PROGRAM MAIN
VAR
		
	bAllDone		: BOOL;
	bStopSequence	: BOOL;
	
	nCase 		: INT;
	nMoveState		: ARRAY[1..nNumMaxMovers] OF INT;
	
	aDynamics	: ARRAY[1..nNumMaxMovers] OF DynamicConstraint_PathXY;
	aMoveOnTrackOptions : ARRAY[1..20] OF ST_MoveOnTrackOptions;
	
	fbXtsEnvironment: FB_TcIoXtsEnvironment;
	
	nForCounter: UDINT;
	M,N,T,Tr,i : UDINT;
	dynamics: INT;
	
	// Magnet
	MagnetValue AT%Q*: INT;
	bMagnetOn : BOOL;	
	stPositionInfo: ST_PositionInfo;
		
	pwm: FB_PWM;
	
	IsMoverCommandedInShortcut: BOOL;
	IsMoverInBlockingArea: BOOL;
	nActStopPos: UINT := 1;
	Fp_error : R_Trig;
	Velo : LREAL := 500;
	Velom1 : LREAL := 500;
	Switch : BOOL;
	WithoutSwitch : BOOL;
	SwtichOnly: BOOL;
	
	MoverStop 		AT%I* : BOOL;
	MoverStopDone 	AT%Q* : BOOL;
	Info 			AT%Q* : BOOL;
	Operating		AT%Q* : BOOL;
	Process			AT%Q* : BOOL;
	Fault			AT%Q* : BOOL;
	Emergency		AT%Q* : BOOL;
	
	Voltage1 		AT%I* : UDINT;
	Voltage2 		AT%I* : UDINT;
	
	
	TcRestart : TC_Restart;
	Restart : BOOL;
	busy : BOOL;
	fp_start : R_Trig;
	bStartSequence: BOOL;
	
	FP_Counter : r_trig;
	Switchcounter : DINT;
	SwitchCurrent: INT :=12; 
	test : LREAL;
	Horntimer : tp; 
	R_trigHorn : R_trig;
	
	TestPowerMat : BOOL;
	StopPos : LREAL := 7611;
	StopTime : TIME := T#8S;
	StopTimer :ARRAY[1..nNumMaxMovers] OF ton;
	StartTimer :ARRAY[1..nNumMaxMovers] OF BOOL;
	
	
	MoverPos :ARRAY[1..nNumMaxMovers] OF PositionXYC;
	ArcLength :ARRAY[1..nNumMaxMovers] OF LREAL;
	TrackPos :ARRAY[1..nNumMaxMovers] OF ARRAY[1..nNumMaxTracks] OF PositionXYC;
	fbFlashlight : Flashlight;
END_VAR

fbXtsEnvironment.Init(TRUE);

Emergency := NOT  MoverStop;


R_trigHorn(clk := MoverStop);
Horntimer(in:= ( R_trigHorn.Q ) , PT:= T#5S,Q=> info);
fbFlashlight(Frequence:=5 , Error=> , Blinker=> );

IF  NOT Horntimer.Q AND MoverStop THEN
	Process := TRUE;
ELSIF Horntimer.Q THEN
	Process:= fbFlashlight.Blinker;
	
ELSE	
	Process := FALSE;
END_IF






IF NOT fbXtsEnvironment.P_IsInitialized THEN
	RETURN;
END_IF

fbXtsEnvironment.XpuTcIo(1).GetPartOids();
IF NOT MoverArrived AND nMoverSartupPos[1].MoverPos <> 0 AND FALSE THEN
	FOR i := 1 TO nNumMaxMovers DO
		fbXtsXlMoverUtility[i].SetConfiguredDetectionTrackObjectId(  nMoverSartupPos[i].TrackID );		
		fbXtsXlMoverUtility[i].SetStartupTrackPosition( (nMoverSartupPos[i].MoverPos)) ;
		fbXtsXlMoverUtility[i].TriggerArrive();
		MoverArrived := TRUE;
	END_FOR	
END_IF



IF NOT MoverStop AND NOT MoverStopDone THEN
	FOR nForCounter:=1 TO nNumMovers DO
		aDynamics[nForCounter].SetValuesVADJ(4000, 4000, 4000, 15000);
		nCase := 140;
		//fbPlanarMover[nForCounter].McPlanarMover.Halt(MoverFeedback[nForCounter], aDynamics[nForCounter]);
	END_FOR		

ELSIF 	MoverStop THEN
	MoverStopDone := FALSE;
END_IF


	TcRestart(
	NETID:= '', 
	RESTART:= Restart, 
	TMOUT:=T#5S , 
	BUSY=>busy , 
	ERR=> , 
	ERRID=> );


fp_start(clk:=bStartSequence);
IF fp_start.Q THEN
	nCase := 10;
	bStartSequence := FALSE;
END_IF


IsMoverCommandedInShortcut := FALSE;
IsMoverInBlockingArea := FALSE;
FOR M := 1 TO nNumMovers DO///Movers
	StopTimer[M](in:=StartTimer[m],PT:=StopTime);
	fbPlanarMover[m].nMoverId := nForCounter;
	fbPlanarMover[m].iTcIoXtsXpuMover := fbXtsEnvironment.XpuTcIo(1).MoverTcIo(TO_UINT(m));
	fbPlanarMover[m].Update();
	
	GVL_mc3.Mover[M].MoverPos :=test :=fbPlanarMover[M].McPlanarMover.MCTOPLC.SETONTRACK.SetPos;
	GVL_mc3.Mover[M].TrackID:= fbPlanarMover[M].McPlanarMover.MCTOPLC.SETONTRACK.TrackOID;
	GVL_mc3.Mover[M].MoverNumber := M;
	
	MoverPos[M].SetValuesXYC(fbPlanarMover[M].McPlanarMover.MCTOPLC.SET.SetPos.x ,fbPlanarMover[M].McPlanarMover.MCTOPLC.SET.SetPos.y,fbPlanarMover[M].McPlanarMover.MCTOPLC.SET.SetPos.c);
	
	TR := Tr+1;
	IF Tr >= nNumMaxTracks THEN
		Tr :=1;
	END_IF
	ArcLength[M] :=GVL_Mc3.MC_Tracks[Tr].GetArcLengthClosestTo(MoverPos[M]);
	GVL_Mc3.MC_Tracks[Tr].GetPositionAt(ArcLength[M],TrackPos[M][Tr]);
	
	IF ABS(MoverPos[m].x - TrackPos[M][Tr].x) < 1 AND  ABS(MoverPos[m].y - TrackPos[M][Tr].y) < 1 THEN
 		GVL_mc3.Mover[M].MoverTrackNr := Tr;
	END_IF	
	
	
		
	IsMoverCommandedInShortcut := IsMoverCommandedInShortcut OR fbPlanarMover[M].IsCommandedInShortcut;
	IsMoverInBlockingArea := IsMoverInBlockingArea OR (Mover[M].TrackID = GVL_Mc3.MC_Tracks[E_TrackNum.main].MCTOPLC_STD.TrackOID AND IsBetween(Mover[M].MoverPos, fMagnetEntry - 100, fMagnetExit + 100));
	MoverFeedback[M].Update();
	
	Fp_error(clk := fbPlanarMover[M].McPlanarMover.Error AND ncase= 100);
	IF Fp_error.Q THEN
		nCase := 140;
		Fault := TRUE;
		bMagnetOn := FALSE;
	
	END_IF
END_FOR

FOR T := 1 TO nNumMaxTracks DO 
	MC_Tracks[T].Update();
	MC_Trackfeedback[T].Update();
	
END_FOR

CASE nCase OF
	10:
		FOR nForCounter := 1 TO fbXtsEnvironment.XpuTcIo(1).GetPartCount() DO
			fbXtsEnvironment.XpuTcIo(1).PartTcIo(TO_UINT(nForCounter)).TriggerReset();
		END_FOR
		Fault := FALSE;
		nCase := 20;

	20:
		FOR T := 1 TO nNumMaxTracks DO 
			MC_Tracks[T].Enable(MC_Trackfeedback[T]);
		END_FOR
				nCase := 30;
		
		
	30: 
		IF MC_Trackfeedback[1].Done AND MC_Trackfeedback[2].Done AND MC_Trackfeedback[3].Done THEN
			nCase := 35;
		END_IF
		
		
	35:
		FOR nForCounter:=1 TO nNumMovers DO
			fbPlanarMover[nForCounter].McPlanarMover.Reset(MoverFeedback[nForCounter]);
		END_FOR
		nCase := 36;	
		
		
	36:	
		bAllDone:=TRUE;
		FOR nForCounter:=1 TO nNumMovers DO
			bAllDone:=bAllDone AND MoverFeedback[nForCounter].Done;
		END_FOR
		
		IF bAllDone THEN
			nCase := 40;
		END_IF
		
		
	40:
		FOR nForCounter:=1 TO nNumMovers DO
			fbPlanarMover[nForCounter].McPlanarMover.Enable(MoverFeedback[nForCounter]);
		END_FOR
		nCase := 50;
	
		
	50:
		bAllDone:=TRUE;
		FOR nForCounter:=1 TO nNumMovers DO
			bAllDone:=bAllDone AND MoverFeedback[nForCounter].Done;
		END_FOR
		
		IF bAllDone THEN
			nCase := 60;
		END_IF

	//55:

	60:
		FOR nForCounter:=nNumMovers TO 1  BY -1 DO
			fbPlanarMover[nForCounter].JoinTrack(MoverFeedback[nForCounter], GVL_Mc3.MC_Tracks[3]);//  Mover[nForCounter].MoverTrackNr]);//
		END_FOR
		
		nCase := 70;
		
		
	70:
		bAllDone:=TRUE;
		FOR nForCounter:=1 TO nNumMovers DO
			bAllDone:=bAllDone AND MoverFeedback[nForCounter].Done;
		END_FOR
		
		IF bAllDone THEN
			nCase := 80;
		END_IF
		
	80:	
		FOR nForCounter:=1 TO nNumMovers DO
			nMoveState[nForCounter] := 0;
			aMoveOnTrackOptions[nForCounter].direction := MC_Direction.mcDirectionPositive;
			aMoveOnTrackOptions[nForCounter].gapMode := MC_GAP_MODE_ON_TRACK.Fast1D;
		END_FOR
		
		nCase := 90;

	100:
		
		FOR nForCounter:=1 TO nNumMovers DO
			aDynamics[nForCounter].SetValuesVADJ(Velo, 4000, 4000, 10000); // (Velo+100, 4000, 4000, 10000); add velo 100 to make a platoon 
			aMoveOnTrackOptions[nForCounter].gap:= 1500; //900 // gap 900 to make a platoon //1500 or 2300 for switches
		END_FOR
	aDynamics[1].SetValuesVADJ(Velo-Velom1, 4000, 4000, 10000);
		FOR nForCounter:=1 TO nNumMovers DO
			CASE nMoveState[nForCounter] OF
				
				0: // Track 3 Main Cycel 
					fbPlanarMover[nForCounter].McPlanarMover.MoveOnTrack(MoverFeedback[nForCounter], GVL_Mc3.MC_Tracks[E_TrackNum.Main],  GVL_Mc3.MC_Tracks[E_TrackNum.Main].GetLength()-1000, aDynamics[nForCounter], aMoveOnTrackOptions[nForCounter]);
					nMoveState[nForCounter] := 10;
					
				10:
					IF Mover[nForCounter].MoverPos > GVL_Mc3.MC_Tracks[E_TrackNum.Main].GetLength()-4000  AND  Mover[nForCounter].TrackID =   GVL_Mc3.MC_Tracks[E_TrackNum.Main].MCTOPLC_STD.TrackOID    THEN//     MCTrackOid_MainSemicircle THEN
						IF (NOT Switch  AND  NOT SwtichOnly) OR WithoutSwitch OR IsMoverCommandedInShortcut THEN
							nMoveState[nForCounter] := 20; // 20 - BigCycel
							IF NOT  WithoutSwitch THEN
								Switch := TRUE;
							ELSE	
								Switch := FALSE;
							END_IF
						ELSE
							nMoveState[nForCounter] := 40;  // 40- SmallCycel
							IsMoverCommandedInShortcut := TRUE;
							Switch := FALSE;
						END_IF
					END_IF

				
				20:
					fbPlanarMover[nForCounter].McPlanarMover.MoveOnTrack(MoverFeedback[nForCounter], GVL_Mc3.MC_Tracks[E_TrackNum.Big], GVL_Mc3.MC_Tracks[E_TrackNum.Big].GetLength()-1000, aDynamics[nForCounter],aMoveOnTrackOptions[nForCounter]);
					nMoveState[nForCounter] := 30;
				
					
				30:
					IF Mover[nForCounter].MoverPos > GVL_Mc3.MC_Tracks[E_TrackNum.Big].GetLength()-4000 AND  Mover[nForCounter].TrackID = GVL_Mc3.MC_Tracks[E_TrackNum.Big].MCTOPLC_STD.TrackOID    THEN//      MCTrackOid_BigSemicircle THEN
						nMoveState[nForCounter] := 60;
					END_IF				
				
			
				40:
					fbPlanarMover[nForCounter].McPlanarMover.MoveOnTrack(MoverFeedback[nForCounter], GVL_Mc3.MC_Tracks[E_TrackNum.Small], (GVL_Mc3.MC_Tracks[E_TrackNum.Small].GetLength()/2), aDynamics[nForCounter], aMoveOnTrackOptions[nForCounter]);
					nMoveState[nForCounter] := 45;	

				45:
					IF MoverFeedback[nForCounter].Done THEN
						fbPlanarMover[nForCounter].McPlanarMover.MoveOnTrack(MoverFeedback[nForCounter], GVL_Mc3.MC_Tracks[E_TrackNum.Small], GVL_Mc3.MC_Tracks[E_TrackNum.Small].GetLength()-1000, aDynamics[nForCounter], aMoveOnTrackOptions[nForCounter]);
						nMoveState[nForCounter] := 50;
					END_IF

			
				50:
					IF Mover[nForCounter].MoverPos > GVL_Mc3.MC_Tracks[E_TrackNum.small].GetLength()-4000 AND  Mover[nForCounter].TrackID = GVL_Mc3.MC_Tracks[E_TrackNum.Small].MCTOPLC_STD.TrackOID    THEN// MCTrackOid_Shortcut THEN
						nMoveState[nForCounter] := 60;
					END_IF
					
				60:
					IF  TestPowerMat  THEN
						nMoveState[nForCounter] := 70;
					ELSE
						nMoveState[nForCounter] := 0;	
					END_IF
				70:
					fbPlanarMover[nForCounter].McPlanarMover.MoveOnTrack(MoverFeedback[nForCounter], GVL_Mc3.MC_Tracks[E_TrackNum.Main], StopPos, aDynamics[nForCounter], aMoveOnTrackOptions[nForCounter]);
					nMoveState[nForCounter] := 80;
				80:
					IF MoverFeedback[nForCounter].Done THEN
						StartTimer[nForCounter] := TRUE;
						nMoveState[nForCounter] := 85;
					END_IF
				85:
					IF 	StopTimer[nForCounter].Q THEN
						StartTimer[nForCounter] := FALSE;
						nMoveState[nForCounter] := 0;	
					END_IF
				END_CASE
		
		END_FOR

		IF bStopSequence AND NOT(IsMoverInBlockingArea) THEN
			nCase := 110;
			bStopSequence := FALSE;
		END_IF
		110:
			N:= nNumMovers;
			FOR nForCounter:=1 TO nNumMovers DO		
				GVL_General.aStopPositions[nForCounter] := TO_LREAL(  fbXtsEnvironment.XpuTcIo(1).MoverTcIo(TO_UINT(N)).GetSimulatedStartUpPosition());
				N := N -1;
			END_FOR
			nCase := 120;
		
		120:	
			nActStopPos := UDINT_TO_UINT(nNumMaxMovers-nNumMovers+1);
			FOR nForCounter:=1 TO nNumMovers DO
				aDynamics[nForCounter].SetValuesVADJ(1000, 4000, 4000, 10000);
				nMoveState[nForCounter] := 0;
				fbPlanarMover[nForCounter].McPlanarMover.MoveOnTrack(MoverFeedback[nForCounter], GVL_Mc3.MC_Tracks[E_TrackNum.main], 300, aDynamics[nForCounter],aMoveOnTrackOptions[nForCounter]);
			END_FOR

			nCase:= 130; 
		130:
			FOR nForCounter:=1 TO nNumMaxMovers - (nNumMaxMovers -nNumMovers)  DO
				CASE nMoveState[nForCounter] OF
					0:								
						
						IF Mover[nForCounter].MoverPos < 300 AND  Mover[nForCounter].TrackID = GVL_Mc3.MC_Tracks[E_TrackNum.main].MCTOPLC_STD.TrackOID THEN
							aMoveOnTrackOptions[nForCounter].gap:= 700;
							fbPlanarMover[nForCounter].McPlanarMover.MoveOnTrack(MoverFeedback[nForCounter], GVL_Mc3.MC_Tracks[E_TrackNum.main], aStopPositions[nActStopPos], aDynamics[nForCounter], aMoveOnTrackOptions[nForCounter]);
							nActStopPos := nActStopPos + 1;
							nMoveState[nForCounter] := 10;
						END_IF
				END_CASE
			END_FOR
		
			bAllDone := TRUE;
			FOR nForCounter:=1 TO nNumMovers DO
				IF NOT(MoverFeedback[nForCounter].Done OR MoverFeedback[nForCounter].Error) THEN
					bAllDone := FALSE;
					EXIT;
				END_IF
			END_FOR
			
			IF bAllDone THEN
				nCase := 150;
			END_IF
		
		140:
			FOR nForCounter:=1 TO nNumMovers DO
				fbPlanarMover[nForCounter].McPlanarMover.Halt(MoverFeedback[nForCounter], aDynamics[nForCounter]);
			END_FOR	
			
			nCase := 145;
			
		145:
			bAllDone := TRUE;
			FOR nForCounter:=1 TO nNumMovers DO
				IF NOT(MoverFeedback[nForCounter].Done OR MoverFeedback[nForCounter].Error) THEN
					bAllDone := FALSE;
					EXIT;
				END_IF
			END_FOR
			
			IF bAllDone THEN
				nCase := 150;
			END_IF
		
		//Disable
		150:
			MoverStopDone := TRUE;
			FOR nForCounter:=1 TO nNumMovers DO
				fbPlanarMover[nForCounter].McPlanarMover.Disable(MoverFeedback[nForCounter]);
			END_FOR
				
			nCase := 0;
END_CASE

bMagnetOn := FALSE;
FOR nForCounter:=1 TO nNumMovers DO
	stPositionInfo := fbXtsEnvironment.XpuTcIo(1).MoverTcIo(TO_UINT(nForCounter)).GetPositionInfo();
	IF stPositionInfo.nTrackObjectId = XtsShortcutOid AND (IsBetween(stPositionInfo.fTrackPosition, fMagnetEntry - (Velo*0.1), fMagnetExit))  THEN
		bMagnetOn := TRUE;
	END_IF
END_FOR

pwm();
	
IF bMagnetOn AND NOT Fault  AND   MoverStop THEN
//Rob July 3 Magnets rescaled 	MagnetValue := SwitchCurrent*1310;
	MagnetValue := SwitchCurrent*2047;  //july 3 scaling, 10V = 16A 
ELSE
 	MagnetValue := 0;
END_IF

FP_Counter(clk:=bMagnetOn);

IF FP_Counter.Q THEN
	Switchcounter := Switchcounter+1;

END_IF

END_PROGRAM

(* stored: Version 1.1.0.1, ProductVersion 3.1.4024.12
   POU MAIN: Id {66ade15a-bef8-4e71-a124-c2e5978c50eb}, SpecialFunc None *)
